// ---- VISUs/v_byte.TcVIS
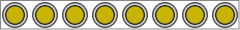
VISUALIZATION v_byte  // 240x30
VAR_IN_OUT
	iNum : INT;
END_VAR
    Lamp1 (0,0 30x30), variable: GVL.stByte.arByte[iNum].Ch[0], style: Lamp-Lamp1-Yellow
    Lamp1 (30,0 30x30), variable: GVL.stByte.arByte[iNum].Ch[1], style: Lamp-Lamp1-Yellow
    Lamp1 (60,0 30x30), variable: GVL.stByte.arByte[iNum].Ch[2], style: Lamp-Lamp1-Yellow
    Lamp1 (90,0 30x30), variable: GVL.stByte.arByte[iNum].Ch[3], style: Lamp-Lamp1-Yellow
    Lamp1 (120,0 30x30), variable: GVL.stByte.arByte[iNum].Ch[4], style: Lamp-Lamp1-Yellow
    Lamp1 (150,0 30x30), variable: GVL.stByte.arByte[iNum].Ch[5], style: Lamp-Lamp1-Yellow
    Lamp1 (180,0 30x30), variable: GVL.stByte.arByte[iNum].Ch[6], style: Lamp-Lamp1-Yellow
    Lamp1 (210,0 30x30), variable: GVL.stByte.arByte[iNum].Ch[7], style: Lamp-Lamp1-Yellow
END_VISUALIZATION

// ---- VISUs/v_IO_ReM.TcVIS
VISUALIZATION v_IO_ReM  // 2048x1080
END_VISUALIZATION

// ---- VISUs/v_rem_0.TcVIS
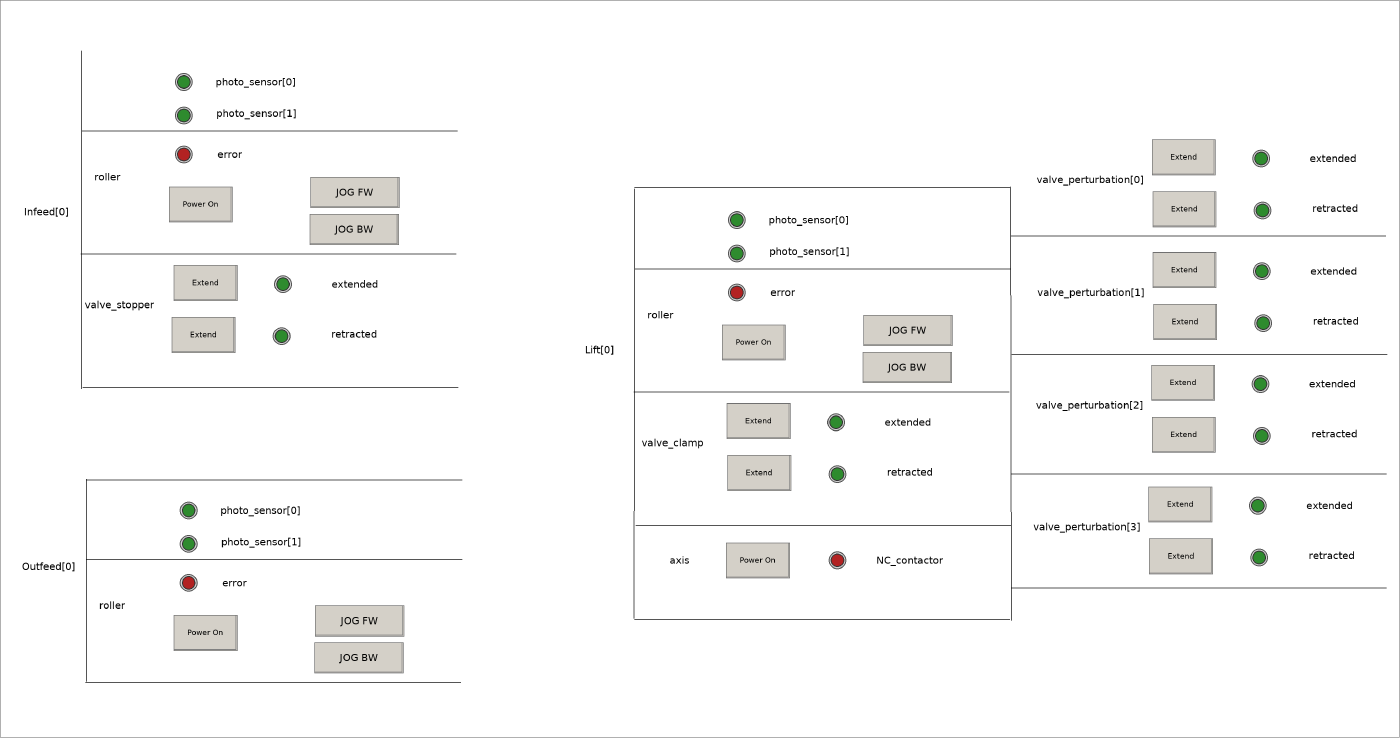
VISUALIZATION v_rem_0  // 2048x1080
VAR_IN_OUT
	dIO_ReM		: Replenishment_Module;
END_VAR
    Lamp1 (254,105 30x30), variable: dIO_ReM.infeed[0].photo_sensor[0].debounced_input.Q, style: Lamp-Lamp1-Green
    Lamp1 (254,154 30x30), variable: dIO_ReM.infeed[0].photo_sensor[1].debounced_input.Q, style: Lamp-Lamp1-Green
    Label (308,107 132x26), "photo_sensor[0]"
    Label (309,153 132x26), "photo_sensor[1]"
    Label (28,297 80x26), "Infeed[0]"
    Lamp1 (254,211 30x30), variable: dIO_ReM.infeed[0].roller.err, style: Lamp-Lamp1-Red
    Label (270,213 132x26), "error"
    Label (91,246 132x26), "roller"
    Line (120,191) (669,191)
    Line (119,74) (119,569)
    Label (109,433 132x26), "valve_stopper"
    Button (454,259 130x45), "JOG FW", colour toggle: dIO_ReM.infeed[0].roller.forward
        OnMouseDown: execute { dIO_ReM.infeed[0].roller.forward := TRUE; }
        OnMouseUp: execute { dIO_ReM.infeed[0].roller.forward := FALSE; }
    Button (453,313 130x45), "JOG BW", colour toggle: dIO_ReM.infeed[0].roller.backward
        OnMouseDown: execute { dIO_ReM.infeed[0].roller.backward := TRUE; }
        OnMouseUp: execute { dIO_ReM.infeed[0].roller.backward := FALSE; }
    Button (247,273 93x52), "Power On", colour toggle: dIO_ReM.infeed[0].roller.Power
        toggle dIO_ReM.infeed[0].roller.Power
    Button (254,388 93x52), "Extend", colour toggle: dIO_ReM.infeed[0].valve_stopper.extend
        OnMouseDown: execute { dIO_ReM.infeed[0].valve_stopper.extend := TRUE; dIO_ReM.infeed[0].valve_stopper.retract := FALSE; }
    Button (251,464 93x52), "Extend", colour toggle: dIO_ReM.infeed[0].valve_stopper.retract
        OnMouseDown: execute { dIO_ReM.infeed[0].valve_stopper.extend := FALSE; dIO_ReM.infeed[0].valve_stopper.retract := TRUE; }
    Lamp1 (399,401 30x30), variable: dIO_ReM.infeed[0].valve_stopper.extended, style: Lamp-Lamp1-Green
    Lamp1 (397,477 30x30), variable: dIO_ReM.infeed[0].valve_stopper.retracted, style: Lamp-Lamp1-Green
    Label (453,403 132x26), "extended"
    Label (452,476 132x26), "retracted"
    Line (118,371) (667,371)
    Line (121,567) (670,567)
    Lamp1 (261,732 30x30), variable: dIO_ReM.outfeed[0].photo_sensor[0].debounced_input.Q, style: Lamp-Lamp1-Green
    Lamp1 (261,781 30x30), variable: dIO_ReM.outfeed[0].photo_sensor[1].debounced_input.Q, style: Lamp-Lamp1-Green
    Label (315,734 132x26), "photo_sensor[0]"
    Label (316,780 132x26), "photo_sensor[1]"
    Label (31,816 80x26), "Outfeed[0]"
    Lamp1 (261,838 30x30), variable: dIO_ReM.outfeed[0].roller.err, style: Lamp-Lamp1-Red
    Label (277,840 132x26), "error"
    Label (98,873 132x26), "roller"
    Line (127,818) (676,818)
    Line (126,701) (126,997)
    Button (461,886 130x45), "JOG FW", colour toggle: dIO_ReM.outfeed[0].roller.forward
        OnMouseDown: execute { dIO_ReM.outfeed[0].roller.forward := TRUE; }
        OnMouseUp: execute { dIO_ReM.outfeed[0].roller.forward := FALSE; }
    Button (460,940 130x45), "JOG BW", colour toggle: dIO_ReM.outfeed[0].roller.backward
        OnMouseDown: execute { dIO_ReM.outfeed[0].roller.backward := TRUE; }
        OnMouseUp: execute { dIO_ReM.outfeed[0].roller.backward := FALSE; }
    Button (254,900 93x52), "Power On", colour toggle: dIO_ReM.outfeed[0].roller.Power
        toggle dIO_ReM.outfeed[0].roller.Power
    Line (125,998) (674,998)
    Line (127,702) (676,702)
    Lamp1 (1063,307 30x30), variable: dIO_ReM.lift[0].photo_sensor[0].debounced_input.Q, style: Lamp-Lamp1-Green
    Lamp1 (1063,356 30x30), variable: dIO_ReM.lift[0].photo_sensor[1].debounced_input.Q, style: Lamp-Lamp1-Green
    Label (1117,309 132x26), "photo_sensor[0]"
    Label (1118,355 132x26), "photo_sensor[1]"
    Label (837,499 80x26), "Lift[0]"
    Lamp1 (1063,413 30x30), variable: dIO_ReM.lift[0].roller.err, style: Lamp-Lamp1-Red
    Label (1079,415 132x26), "error"
    Label (900,448 132x26), "roller"
    Line (929,393) (1478,393)
    Line (928,276) (927,905)
    Label (918,635 132x26), "valve_clamp"
    Button (1263,461 130x45), "JOG FW", colour toggle: dIO_ReM.lift[0].roller.forward
        OnMouseDown: execute { dIO_ReM.lift[0].roller.forward := TRUE; }
        OnMouseUp: execute { dIO_ReM.lift[0].roller.forward := FALSE; }
    Button (1262,515 130x45), "JOG BW", colour toggle: dIO_ReM.lift[0].roller.backward
        OnMouseDown: execute { dIO_ReM.lift[0].roller.backward := TRUE; }
        OnMouseUp: execute { dIO_ReM.lift[0].roller.backward := FALSE; }
    Button (1056,475 93x52), "Power On", colour toggle: dIO_ReM.lift[0].roller.Power
        toggle dIO_ReM.lift[0].roller.Power
    Button (1063,590 93x52), "Extend", colour toggle: dIO_ReM.lift[0].valve_clamp.extend
        OnMouseDown: execute { dIO_ReM.lift[0].valve_clamp.extend := TRUE; dIO_ReM.lift[0].valve_clamp.retract := FALSE; }
    Button (1064,666 93x52), "Extend", colour toggle: dIO_ReM.lift[0].valve_clamp.retract
        OnMouseDown: execute { dIO_ReM.lift[0].valve_clamp.extend := FALSE; dIO_ReM.lift[0].valve_clamp.retract := TRUE; }
    Lamp1 (1208,603 30x30), variable: dIO_ReM.lift[0].valve_clamp.extended, style: Lamp-Lamp1-Green
    Lamp1 (1210,679 30x30), variable: dIO_ReM.lift[0].valve_clamp.retracted, style: Lamp-Lamp1-Green
    Label (1262,605 132x26), "extended"
    Label (1265,678 132x26), "retracted"
    Line (927,573) (1476,573)
    Line (930,769) (1479,769)
    Label (1515,250 160x26), "valve_perturbation[0]"
    Button (1685,204 93x52), "Extend", colour toggle: dIO_ReM.lift[0].valve_perturbation[0].extend
        OnMouseDown: execute { dIO_ReM.lift[0].valve_perturbation[0].extend := TRUE; dIO_ReM.lift[0].valve_perturbation[0].retract := FALSE; }
    Button (1686,280 93x52), "Extend", colour toggle: dIO_ReM.lift[0].valve_perturbation[0].retract
        OnMouseDown: execute { dIO_ReM.lift[0].valve_perturbation[0].extend := FALSE; dIO_ReM.lift[0].valve_perturbation[0].retract := TRUE; }
    Lamp1 (1830,217 30x30), variable: dIO_ReM.lift[0].valve_perturbation[0].extended, style: Lamp-Lamp1-Green
    Lamp1 (1832,293 30x30), variable: dIO_ReM.lift[0].valve_perturbation[0].retracted, style: Lamp-Lamp1-Green
    Label (1884,219 132x26), "extended"
    Label (1887,292 132x26), "retracted"
    Label (1516,415 160x26), "valve_perturbation[1]"
    Button (1686,369 93x52), "Extend", colour toggle: dIO_ReM.lift[0].valve_perturbation[1].extend
        OnMouseDown: execute { dIO_ReM.lift[0].valve_perturbation[1].extend := TRUE; dIO_ReM.lift[0].valve_perturbation[1].retract := FALSE; }
    Button (1687,445 93x52), "Extend", colour toggle: dIO_ReM.lift[0].valve_perturbation[1].retract
        OnMouseDown: execute { dIO_ReM.lift[0].valve_perturbation[1].extend := FALSE; dIO_ReM.lift[0].valve_perturbation[1].retract := TRUE; }
    Lamp1 (1831,382 30x30), variable: dIO_ReM.lift[0].valve_perturbation[1].extended, style: Lamp-Lamp1-Green
    Lamp1 (1833,458 30x30), variable: dIO_ReM.lift[0].valve_perturbation[1].retracted, style: Lamp-Lamp1-Green
    Label (1885,384 132x26), "extended"
    Label (1888,457 132x26), "retracted"
    Label (1514,580 160x26), "valve_perturbation[2]"
    Button (1684,534 93x52), "Extend", colour toggle: dIO_ReM.lift[0].valve_perturbation[2].extend
        OnMouseDown: execute { dIO_ReM.lift[0].valve_perturbation[2].extend := TRUE; dIO_ReM.lift[0].valve_perturbation[2].retract := FALSE; }
    Button (1685,610 93x52), "Extend", colour toggle: dIO_ReM.lift[0].valve_perturbation[2].retract
        OnMouseDown: execute { dIO_ReM.lift[0].valve_perturbation[2].extend := FALSE; dIO_ReM.lift[0].valve_perturbation[2].retract := TRUE; }
    Lamp1 (1829,547 30x30), variable: dIO_ReM.lift[0].valve_perturbation[2].extended, style: Lamp-Lamp1-Green
    Lamp1 (1831,623 30x30), variable: dIO_ReM.lift[0].valve_perturbation[2].retracted, style: Lamp-Lamp1-Green
    Label (1883,549 132x26), "extended"
    Label (1886,622 132x26), "retracted"
    Label (1510,758 160x26), "valve_perturbation[3]"
    Button (1680,712 93x52), "Extend", colour toggle: dIO_ReM.lift[0].valve_perturbation[3].extend
        OnMouseDown: execute { dIO_ReM.lift[0].valve_perturbation[3].extend := TRUE; dIO_ReM.lift[0].valve_perturbation[3].retract := FALSE; }
    Button (1681,788 93x52), "Extend", colour toggle: dIO_ReM.lift[0].valve_perturbation[3].retract
        OnMouseDown: execute { dIO_ReM.lift[0].valve_perturbation[3].extend := FALSE; dIO_ReM.lift[0].valve_perturbation[3].retract := TRUE; }
    Lamp1 (1825,725 30x30), variable: dIO_ReM.lift[0].valve_perturbation[3].extended, style: Lamp-Lamp1-Green
    Lamp1 (1827,801 30x30), variable: dIO_ReM.lift[0].valve_perturbation[3].retracted, style: Lamp-Lamp1-Green
    Label (1879,727 132x26), "extended"
    Label (1882,800 132x26), "retracted"
    Line (1478,273) (1479,908)
    Line (1478,345) (2027,345)
    Line (1480,518) (2029,518)
    Line (1479,693) (2028,693)
    Line (1479,860) (2028,860)
    Line (928,274) (1477,274)
    Line (928,906) (1477,906)
    Label (1265,807 132x26), "NC_contactor"
    Label (928,807 132x26), "axis"
    Button (1062,794 93x52), "Power On", colour toggle: dIO_ReM.lift[0].power_axis
        toggle dIO_ReM.lift[0].power_axis
    Lamp1 (1210,805 30x30), variable: dIO_ReM.lift[0].contactor_axis, style: Lamp-Lamp1-Red
END_VISUALIZATION

// ---- VISUs/v_pm_0.TcVIS
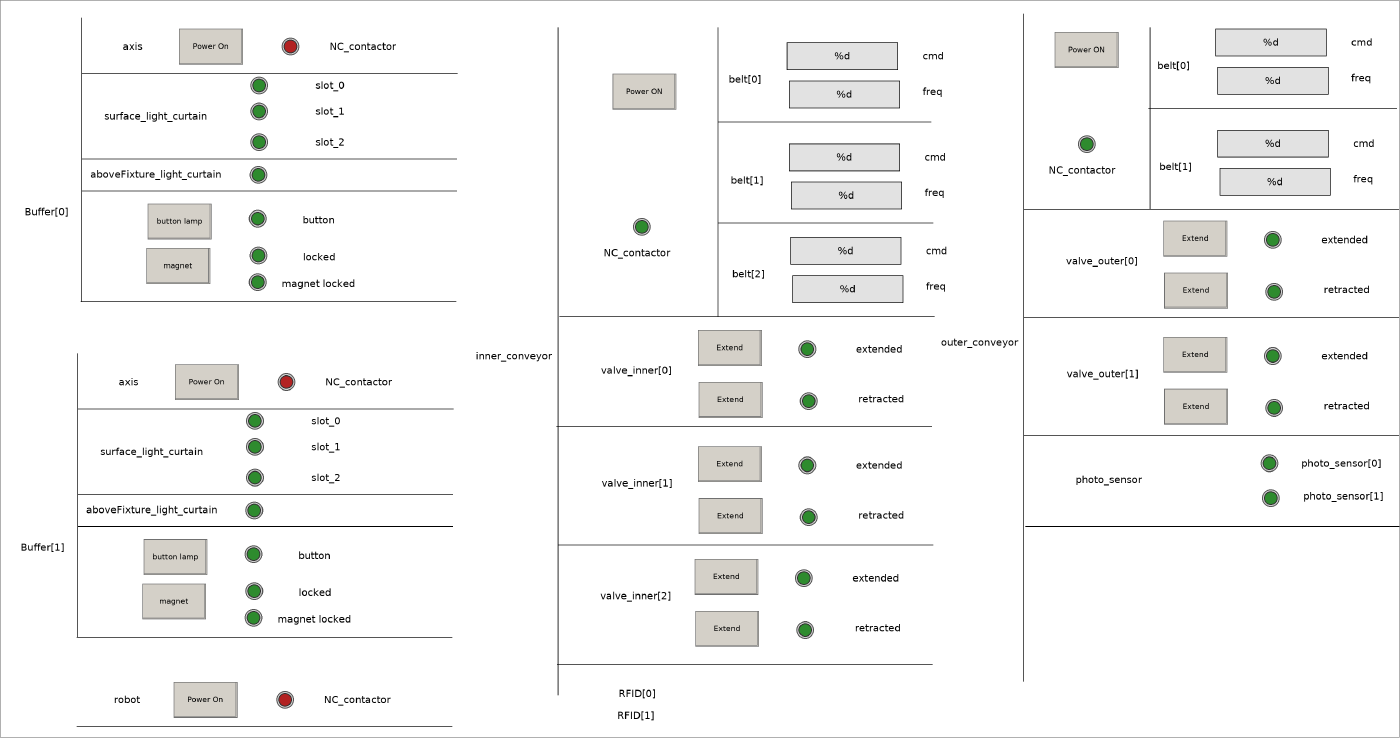
VISUALIZATION v_pm_0  // 2048x1080
VAR_IN_OUT
	dIO_PM		: Picking_Module;
END_VAR
    Lamp1 (364,110 30x30), variable: dIO_PM.buffer[0].surfae_slot_0, style: Lamp-Lamp1-Green
    Label (418,112 130x26), "slot_0"
    Label (28,297 80x26), "Buffer[0]"
    Line (120,107) (669,107)
    Line (119,26) (119,441)
    Line (118,441) (667,441)
    Label (672,508 160x26), "inner_conveyor"
    Line (816,40) (816,1017)
    Label (851,529 160x26), "valve_inner[0]"
    Button (1021,483 93x52), "Extend", colour toggle: dIO_PM.inConv.valve[0].extend
        OnMouseDown: execute { dIO_PM.inConv.valve[0].extend := TRUE; dIO_PM.inConv.valve[0].retract := FALSE; }
    Button (1022,559 93x52), "Extend", colour toggle: dIO_PM.inConv.valve[0].retract
        OnMouseDown: execute { dIO_PM.inConv.valve[0].extend := FALSE; dIO_PM.inConv.valve[0].retract := TRUE; }
    Lamp1 (1166,496 30x30), variable: dIO_PM.inConv.valve[0].extended, style: Lamp-Lamp1-Green
    Lamp1 (1168,572 30x30), variable: dIO_PM.inConv.valve[0].retracted, style: Lamp-Lamp1-Green
    Label (1220,498 132x26), "extended"
    Label (1223,571 132x26), "retracted"
    Label (852,694 160x26), "valve_inner[1]"
    Label (850,859 160x26), "valve_inner[2]"
    Line (814,624) (1363,624)
    Line (816,797) (1365,797)
    Line (815,972) (1364,972)
    Label (465,55 132x26), "NC_contactor"
    Label (128,55 132x26), "axis"
    Button (262,42 93x52), "Power On", colour toggle: dIO_PM.buffer[0].power_axis
        toggle dIO_PM.buffer[0].power_axis
    Lamp1 (410,53 30x30), variable: dIO_PM.buffer[0].contractor_axis, style: Lamp-Lamp1-Red
    Label (128,157 200x26), "surface_light_curtain"
    Label (418,150 130x26), "slot_1"
    Lamp1 (364,148 30x30), variable: dIO_PM.buffer[0].surfae_slot_1, style: Lamp-Lamp1-Green
    Label (418,195 130x26), "slot_2"
    Lamp1 (364,193 30x30), variable: dIO_PM.buffer[0].surfae_slot_2, style: Lamp-Lamp1-Green
    Label (128,242 200x26), "aboveFixture_light_curtain"
    Lamp1 (363,241 30x30), variable: dIO_PM.buffer[0].above_fixture_light_curtain, style: Lamp-Lamp1-Green
    Line (119,232) (668,232)
    Line (119,279) (668,279)
    Label (406,309 120x26), "button"
    Lamp1 (362,305 30x30), variable: dIO_PM.buffer[0].button, style: Lamp-Lamp1-Green
    Button (216,298 93x52), "button lamp", colour toggle: dIO_PM.buffer[0].lamp_button
        toggle dIO_PM.buffer[0].lamp_button
    Button (214,363 93x52), "magnet", colour toggle: dIO_PM.buffer[0].magnet
        toggle dIO_PM.buffer[0].magnet
    Label (407,363 120x26), "locked"
    Lamp1 (363,359 30x30), variable: dIO_PM.buffer[0].locked, style: Lamp-Lamp1-Green
    Label (406,402 120x26), "magnet locked"
    Lamp1 (362,398 30x30), variable: dIO_PM.buffer[0].magnet_locked, style: Lamp-Lamp1-Green
    Lamp1 (358,601 30x30), variable: dIO_PM.buffer[1].surfae_slot_0, style: Lamp-Lamp1-Green
    Label (412,603 130x26), "slot_0"
    Label (22,788 80x26), "Buffer[1]"
    Line (114,598) (663,598)
    Line (113,517) (113,932)
    Line (112,932) (661,932)
    Label (459,546 132x26), "NC_contactor"
    Label (122,546 132x26), "axis"
    Button (256,533 93x52), "Power On", colour toggle: dIO_PM.buffer[1].power_axis
        toggle dIO_PM.buffer[1].power_axis
    Lamp1 (404,544 30x30), variable: dIO_PM.buffer[1].contractor_axis, style: Lamp-Lamp1-Red
    Label (122,648 200x26), "surface_light_curtain"
    Label (412,641 130x26), "slot_1"
    Lamp1 (358,639 30x30), variable: dIO_PM.buffer[1].surfae_slot_1, style: Lamp-Lamp1-Green
    Label (412,686 130x26), "slot_2"
    Lamp1 (358,684 30x30), variable: dIO_PM.buffer[1].surfae_slot_2, style: Lamp-Lamp1-Green
    Label (122,733 200x26), "aboveFixture_light_curtain"
    Lamp1 (357,732 30x30), variable: dIO_PM.buffer[1].above_fixture_light_curtain, style: Lamp-Lamp1-Green
    Line (113,723) (662,723)
    Line (113,770) (662,770)
    Label (400,800 120x26), "button"
    Lamp1 (356,796 30x30), variable: dIO_PM.buffer[1].button, style: Lamp-Lamp1-Green
    Button (210,789 93x52), "button lamp", colour toggle: dIO_PM.buffer[0].lamp_button
        toggle dIO_PM.buffer[1].lamp_button
    Button (208,854 93x52), "magnet", colour toggle: dIO_PM.buffer[1].magnet
        toggle dIO_PM.buffer[1].magnet
    Label (401,854 120x26), "locked"
    Lamp1 (357,850 30x30), variable: dIO_PM.buffer[1].locked, style: Lamp-Lamp1-Green
    Label (400,893 120x26), "magnet locked"
    Lamp1 (356,889 30x30), variable: dIO_PM.buffer[1].magnet_locked, style: Lamp-Lamp1-Green
    Line (112,1063) (661,1063)
    Label (457,1011 132x26), "NC_contactor"
    Label (120,1011 132x26), "robot"
    Button (254,998 93x52), "Power On", colour toggle: dIO_PM.power_robot
        toggle dIO_PM.power_robot
    Lamp1 (402,1009 30x30), variable: dIO_PM.contactor_robot, style: Lamp-Lamp1-Red
    Rectangle (1151,62 162x40), "%d", text variable: dIO_PM.inConv.belt[0].cmd
        OnMouseClick: write the text variable via Default
    Rectangle (1154,118 162x40), "%d", text variable: dIO_PM.inConv.belt[0].freq
        OnMouseClick: write the text variable via Default
    Label (1024,103 132x26), "belt[0]"
    Label (1299,69 132x26), "cmd"
    Label (1298,121 132x26), "freq"
    Line (1050,178) (1362,178)
    Rectangle (1154,210 162x40), "%d", text variable: dIO_PM.inConv.belt[1].cmd
        OnMouseClick: write the text variable via Default
    Rectangle (1157,266 162x40), "%d", text variable: dIO_PM.inConv.belt[1].freq
        OnMouseClick: write the text variable via Default
    Label (1027,251 132x26), "belt[1]"
    Label (1302,217 132x26), "cmd"
    Label (1301,269 132x26), "freq"
    Line (1050,326) (1365,326)
    Rectangle (1156,347 162x40), "%d", text variable: dIO_PM.inConv.belt[2].cmd
        OnMouseClick: write the text variable via Default
    Rectangle (1159,403 162x40), "%d", text variable: dIO_PM.inConv.belt[2].freq
        OnMouseClick: write the text variable via Default
    Label (1029,388 132x26), "belt[2]"
    Label (1304,354 132x26), "cmd"
    Label (1303,406 132x26), "freq"
    Line (818,463) (1367,463)
    Button (1021,653 93x52), "Extend", colour toggle: dIO_PM.inConv.valve[1].extend
        OnMouseDown: execute { dIO_PM.inConv.valve[1].extend := TRUE; dIO_PM.inConv.valve[1].retract := FALSE; }
    Button (1022,729 93x52), "Extend", colour toggle: dIO_PM.inConv.valve[1].retract
        OnMouseDown: execute { dIO_PM.inConv.valve[1].extend := FALSE; dIO_PM.inConv.valve[1].retract := TRUE; }
    Lamp1 (1166,666 30x30), variable: dIO_PM.inConv.valve[1].extended, style: Lamp-Lamp1-Green
    Lamp1 (1168,742 30x30), variable: dIO_PM.inConv.valve[1].retracted, style: Lamp-Lamp1-Green
    Label (1220,668 132x26), "extended"
    Label (1223,741 132x26), "retracted"
    Button (1016,818 93x52), "Extend", colour toggle: dIO_PM.inConv.valve[2].extend
        OnMouseDown: execute { dIO_PM.inConv.valve[2].extend := TRUE; dIO_PM.inConv.valve[2].retract := FALSE; }
    Button (1017,894 93x52), "Extend", colour toggle: dIO_PM.inConv.valve[2].retract
        OnMouseDown: execute { dIO_PM.inConv.valve[2].extend := FALSE; dIO_PM.inConv.valve[2].retract := TRUE; }
    Lamp1 (1161,831 30x30), variable: dIO_PM.inConv.valve[2].extended, style: Lamp-Lamp1-Green
    Lamp1 (1163,907 30x30), variable: dIO_PM.inConv.valve[2].retracted, style: Lamp-Lamp1-Green
    Label (1215,833 132x26), "extended"
    Label (1218,906 132x26), "retracted"
    Label (852,1002 160x26), "RFID[0]"
    Label (850,1034 160x26), "RFID[1]"
    Label (1353,488 160x26), "outer_conveyor"
    Line (1497,20) (1497,997)
    Label (1532,369 160x26), "valve_outer[0]"
    Button (1702,323 93x52), "Extend", colour toggle: dIO_PM.outConv.valve[0].extend
        OnMouseDown: execute { dIO_PM.outConv.valve[0].extend := TRUE; dIO_PM.outConv.valve[0].retract := FALSE; }
    Button (1703,399 93x52), "Extend", colour toggle: dIO_PM.outConv.valve[0].retract
        OnMouseDown: execute { dIO_PM.outConv.valve[0].extend := FALSE; dIO_PM.outConv.valve[0].retract := TRUE; }
    Lamp1 (1847,336 30x30), variable: dIO_PM.outConv.valve[0].extended, style: Lamp-Lamp1-Green
    Lamp1 (1849,412 30x30), variable: dIO_PM.outConv.valve[0].retracted, style: Lamp-Lamp1-Green
    Label (1901,338 132x26), "extended"
    Label (1904,411 132x26), "retracted"
    Label (1533,534 160x26), "valve_outer[1]"
    Line (1498,464) (2047,464)
    Line (1497,637) (2046,637)
    Line (1500,770) (2049,770)
    Rectangle (1778,42 162x40), "%d", text variable: dIO_PM.outConv.belt[0].cmd
        OnMouseClick: write the text variable via Default
    Rectangle (1781,98 162x40), "%d", text variable: dIO_PM.outConv.belt[0].freq
        OnMouseClick: write the text variable via Default
    Label (1651,83 132x26), "belt[0]"
    Label (1926,49 132x26), "cmd"
    Label (1925,101 132x26), "freq"
    Line (1680,158) (2043,158)
    Rectangle (1781,190 162x40), "%d", text variable: dIO_PM.outConv.belt[1].cmd
        OnMouseClick: write the text variable via Default
    Rectangle (1784,246 162x40), "%d", text variable: dIO_PM.outConv.belt[1].freq
        OnMouseClick: write the text variable via Default
    Label (1654,231 132x26), "belt[1]"
    Label (1929,197 132x26), "cmd"
    Label (1928,249 132x26), "freq"
    Line (1497,306) (2046,306)
    Button (1702,493 93x52), "Extend", colour toggle: dIO_PM.outConv.valve[1].extend
        OnMouseDown: execute { dIO_PM.outConv.valve[1].extend := TRUE; dIO_PM.outConv.valve[1].retract := FALSE; }
    Button (1703,569 93x52), "Extend", colour toggle: dIO_PM.outConv.valve[1].retract
        OnMouseDown: execute { dIO_PM.outConv.valve[1].extend := FALSE; dIO_PM.outConv.valve[1].retract := TRUE; }
    Lamp1 (1847,506 30x30), variable: dIO_PM.outConv.valve[1].extended, style: Lamp-Lamp1-Green
    Lamp1 (1849,582 30x30), variable: dIO_PM.outConv.valve[1].retracted, style: Lamp-Lamp1-Green
    Label (1901,508 132x26), "extended"
    Label (1904,581 132x26), "retracted"
    Lamp1 (1842,663 30x30), variable: dIO_PM.outConv.photo_sensor[0], style: Lamp-Lamp1-Green
    Lamp1 (1844,714 30x30), variable: dIO_PM.outConv.photo_sensor[1], style: Lamp-Lamp1-Green
    Label (1896,665 132x26), "photo_sensor[0]"
    Label (1899,713 132x26), "photo_sensor[1]"
    Label (1542,689 160x26), "photo_sensor"
    Line (1050,40) (1050,463)
    Button (896,108 93x52), "Power ON", colour toggle: dIO_PM.power_inConv
        toggle dIO_PM.power_inConv
    Lamp1 (924,317 30x30), variable: dIO_PM.contactor_inConv, style: Lamp-Lamp1-Green
    Label (866,357 132x26), "NC_contactor"
    Line (1682,40) (1682,306)
    Button (1543,47 93x52), "Power ON", colour toggle: dIO_PM.power_outConv
        toggle dIO_PM.power_outConv
    Lamp1 (1575,196 30x30), variable: dIO_PM.contactor_outConv, style: Lamp-Lamp1-Green
    Label (1517,236 132x26), "NC_contactor"
END_VISUALIZATION

// ---- VISUs/v_rem_1.TcVIS
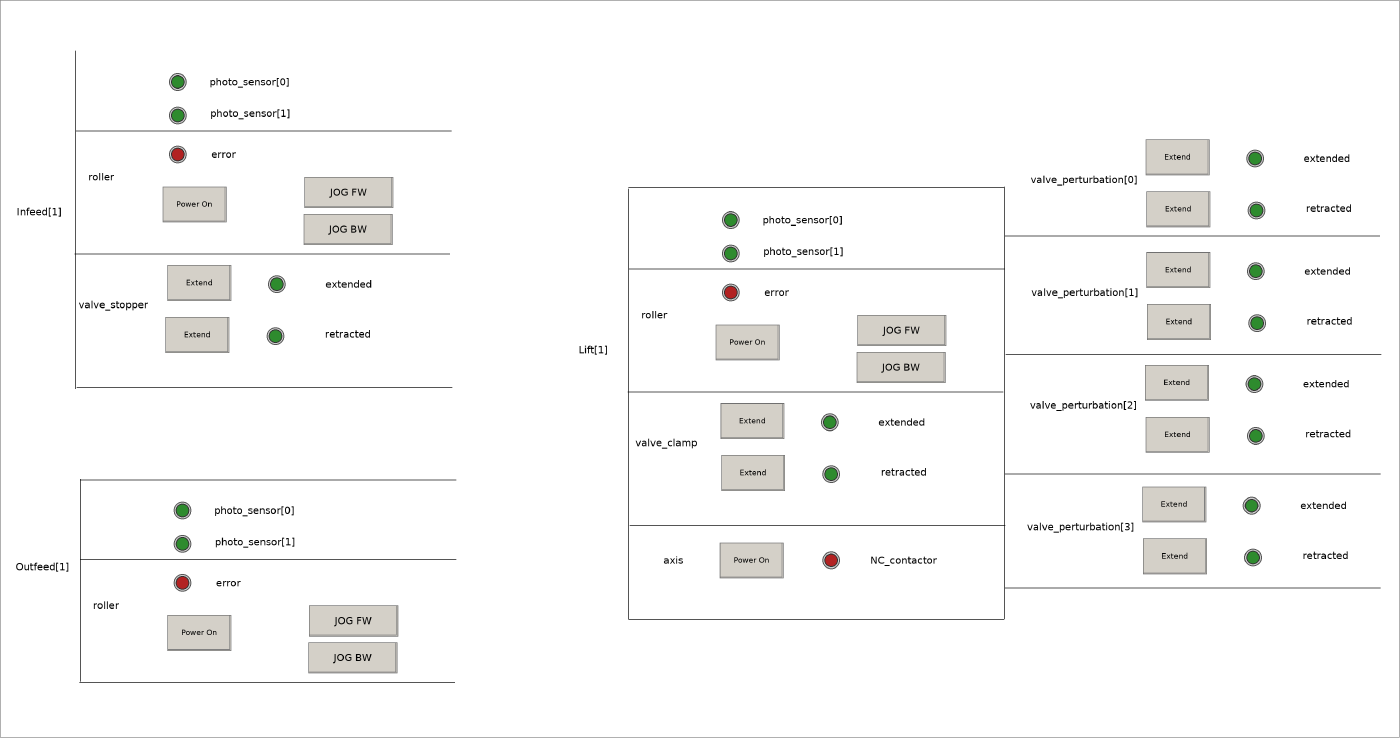
VISUALIZATION v_rem_1  // 2048x1080
VAR_IN_OUT
	dIO_ReM		: Replenishment_Module;
END_VAR
    Lamp1 (245,105 30x30), variable: dIO_ReM.infeed[1].photo_sensor[0].debounced_input.Q, style: Lamp-Lamp1-Green
    Lamp1 (245,154 30x30), variable: dIO_ReM.infeed[1].photo_sensor[1].debounced_input.Q, style: Lamp-Lamp1-Green
    Label (299,107 132x26), "photo_sensor[0]"
    Label (300,153 132x26), "photo_sensor[1]"
    Label (19,297 77x26), "Infeed[1]"
    Lamp1 (245,211 30x30), variable: dIO_ReM.infeed[1].roller.err, style: Lamp-Lamp1-Red
    Label (261,213 132x26), "error"
    Label (82,246 132x26), "roller"
    Line (111,191) (660,191)
    Line (110,74) (110,569)
    Label (100,433 132x26), "valve_stopper"
    Button (445,259 130x45), "JOG FW", colour toggle: dIO_ReM.infeed[1].roller.forward
        OnMouseDown: execute { dIO_ReM.infeed[1].roller.forward := TRUE; }
        OnMouseUp: execute { dIO_ReM.infeed[1].roller.forward := FALSE; }
    Button (444,313 130x45), "JOG BW", colour toggle: dIO_ReM.infeed[1].roller.backward
        OnMouseDown: execute { dIO_ReM.infeed[1].roller.backward := TRUE; }
        OnMouseUp: execute { dIO_ReM.infeed[1].roller.backward := FALSE; }
    Button (238,273 93x52), "Power On", colour toggle: dIO_ReM.infeed[1].roller.Power
        toggle dIO_ReM.infeed[1].roller.Power
    Button (245,388 93x52), "Extend", colour toggle: dIO_ReM.infeed[1].valve_stopper.extend
        OnMouseDown: execute { dIO_ReM.infeed[1].valve_stopper.extend := TRUE; dIO_ReM.infeed[1].valve_stopper.retract := FALSE; }
    Button (242,464 93x52), "Extend", colour toggle: dIO_ReM.infeed[1].valve_stopper.retract
        OnMouseDown: execute { dIO_ReM.infeed[1].valve_stopper.extend := FALSE; dIO_ReM.infeed[1].valve_stopper.retract := TRUE; }
    Lamp1 (390,401 30x30), variable: dIO_ReM.infeed[1].valve_stopper.extended, style: Lamp-Lamp1-Green
    Lamp1 (388,477 30x30), variable: dIO_ReM.infeed[1].valve_stopper.retracted, style: Lamp-Lamp1-Green
    Label (444,403 132x26), "extended"
    Label (443,476 132x26), "retracted"
    Line (109,371) (658,371)
    Line (112,567) (661,567)
    Lamp1 (252,732 30x30), variable: dIO_ReM.outfeed[1].photo_sensor[0].debounced_input.Q, style: Lamp-Lamp1-Green
    Lamp1 (252,781 30x30), variable: dIO_ReM.outfeed[1].photo_sensor[1].debounced_input.Q, style: Lamp-Lamp1-Green
    Label (306,734 132x26), "photo_sensor[0]"
    Label (307,780 132x26), "photo_sensor[1]"
    Label (22,816 80x27), "Outfeed[1]"
    Lamp1 (252,838 30x30), variable: dIO_ReM.outfeed[1].roller.err, style: Lamp-Lamp1-Red
    Label (268,840 132x26), "error"
    Label (89,873 132x26), "roller"
    Line (118,818) (667,818)
    Line (117,701) (117,997)
    Button (452,886 130x45), "JOG FW", colour toggle: dIO_ReM.outfeed[1].roller.forward
        OnMouseDown: execute { dIO_ReM.outfeed[1].roller.forward := TRUE; }
        OnMouseUp: execute { dIO_ReM.outfeed[1].roller.forward := FALSE; }
    Button (451,940 130x45), "JOG BW", colour toggle: dIO_ReM.outfeed[1].roller.backward
        OnMouseDown: execute { dIO_ReM.outfeed[1].roller.backward := TRUE; }
        OnMouseUp: execute { dIO_ReM.outfeed[1].roller.backward := FALSE; }
    Button (245,900 93x52), "Power On", colour toggle: dIO_ReM.outfeed[1].roller.Power
        toggle dIO_ReM.outfeed[1].roller.Power
    Line (116,998) (665,998)
    Line (118,702) (667,702)
    Lamp1 (1054,307 30x30), variable: dIO_ReM.lift[1].photo_sensor[0].debounced_input.Q, style: Lamp-Lamp1-Green
    Lamp1 (1054,356 30x30), variable: dIO_ReM.lift[1].photo_sensor[1].debounced_input.Q, style: Lamp-Lamp1-Green
    Label (1108,309 132x26), "photo_sensor[0]"
    Label (1109,355 132x26), "photo_sensor[1]"
    Label (828,499 80x26), "Lift[1]"
    Lamp1 (1054,413 30x30), variable: dIO_ReM.lift[1].roller.err, style: Lamp-Lamp1-Red
    Label (1070,415 132x26), "error"
    Label (891,448 132x26), "roller"
    Line (920,393) (1469,393)
    Line (919,276) (919,906)
    Label (909,635 132x26), "valve_clamp"
    Button (1254,461 130x45), "JOG FW", colour toggle: dIO_ReM.lift[1].roller.forward
        OnMouseDown: execute { dIO_ReM.lift[1].roller.forward := TRUE; }
        OnMouseUp: execute { dIO_ReM.lift[1].roller.forward := FALSE; }
    Button (1253,515 130x45), "JOG BW", colour toggle: dIO_ReM.lift[1].roller.backward
        OnMouseDown: execute { dIO_ReM.lift[1].roller.backward := TRUE; }
        OnMouseUp: execute { dIO_ReM.lift[1].roller.backward := FALSE; }
    Button (1047,475 93x52), "Power On", colour toggle: dIO_ReM.lift[1].roller.Power
        toggle dIO_ReM.lift[1].roller.Power
    Button (1054,590 93x52), "Extend", colour toggle: dIO_ReM.lift[1].valve_clamp.extend
        OnMouseDown: execute { dIO_ReM.lift[1].valve_clamp.extend := TRUE; dIO_ReM.lift[1].valve_clamp.retract := FALSE; }
    Button (1055,666 93x52), "Extend", colour toggle: dIO_ReM.lift[1].valve_clamp.retract
        OnMouseDown: execute { dIO_ReM.lift[1].valve_clamp.extend := FALSE; dIO_ReM.lift[1].valve_clamp.retract := TRUE; }
    Lamp1 (1199,603 30x30), variable: dIO_ReM.lift[1].valve_clamp.extended, style: Lamp-Lamp1-Green
    Lamp1 (1201,679 30x30), variable: dIO_ReM.lift[1].valve_clamp.retracted, style: Lamp-Lamp1-Green
    Label (1253,605 132x26), "extended"
    Label (1256,678 132x26), "retracted"
    Line (918,573) (1467,573)
    Line (921,769) (1470,769)
    Label (1506,250 160x26), "valve_perturbation[0]"
    Button (1676,204 93x52), "Extend", colour toggle: dIO_ReM.lift[1].valve_perturbation[0].extend
        OnMouseDown: execute { dIO_ReM.lift[1].valve_perturbation[0].extend := TRUE; dIO_ReM.lift[1].valve_perturbation[0].retract := FALSE; }
    Button (1677,280 93x52), "Extend", colour toggle: dIO_ReM.lift[1].valve_perturbation[0].retract
        OnMouseDown: execute { dIO_ReM.lift[1].valve_perturbation[0].extend := FALSE; dIO_ReM.lift[1].valve_perturbation[0].retract := TRUE; }
    Lamp1 (1821,217 30x30), variable: dIO_ReM.lift[1].valve_perturbation[0].extended, style: Lamp-Lamp1-Green
    Lamp1 (1823,293 30x30), variable: dIO_ReM.lift[1].valve_perturbation[0].retracted, style: Lamp-Lamp1-Green
    Label (1875,219 132x26), "extended"
    Label (1878,292 132x26), "retracted"
    Label (1507,415 160x26), "valve_perturbation[1]"
    Button (1677,369 93x52), "Extend", colour toggle: dIO_ReM.lift[1].valve_perturbation[1].extend
        OnMouseDown: execute { dIO_ReM.lift[1].valve_perturbation[1].extend := TRUE; dIO_ReM.lift[1].valve_perturbation[1].retract := FALSE; }
    Button (1678,445 93x52), "Extend", colour toggle: dIO_ReM.lift[1].valve_perturbation[1].retract
        OnMouseDown: execute { dIO_ReM.lift[1].valve_perturbation[1].extend := FALSE; dIO_ReM.lift[1].valve_perturbation[1].retract := TRUE; }
    Lamp1 (1822,382 30x30), variable: dIO_ReM.lift[1].valve_perturbation[1].extended, style: Lamp-Lamp1-Green
    Lamp1 (1824,458 30x30), variable: dIO_ReM.lift[1].valve_perturbation[1].retracted, style: Lamp-Lamp1-Green
    Label (1876,384 132x26), "extended"
    Label (1879,457 132x26), "retracted"
    Label (1505,580 160x26), "valve_perturbation[2]"
    Button (1675,534 93x52), "Extend", colour toggle: dIO_ReM.lift[1].valve_perturbation[2].extend
        OnMouseDown: execute { dIO_ReM.lift[1].valve_perturbation[2].extend := TRUE; dIO_ReM.lift[1].valve_perturbation[2].retract := FALSE; }
    Button (1676,610 93x52), "Extend", colour toggle: dIO_ReM.lift[1].valve_perturbation[2].retract
        OnMouseDown: execute { dIO_ReM.lift[1].valve_perturbation[2].extend := FALSE; dIO_ReM.lift[1].valve_perturbation[2].retract := TRUE; }
    Lamp1 (1820,547 30x30), variable: dIO_ReM.lift[1].valve_perturbation[2].extended, style: Lamp-Lamp1-Green
    Lamp1 (1822,623 30x30), variable: dIO_ReM.lift[1].valve_perturbation[2].retracted, style: Lamp-Lamp1-Green
    Label (1874,549 132x26), "extended"
    Label (1877,622 132x26), "retracted"
    Label (1501,758 160x26), "valve_perturbation[3]"
    Button (1671,712 93x52), "Extend", colour toggle: dIO_ReM.lift[1].valve_perturbation[3].extend
        OnMouseDown: execute { dIO_ReM.lift[1].valve_perturbation[3].extend := TRUE; dIO_ReM.lift[1].valve_perturbation[3].retract := FALSE; }
    Button (1672,788 93x52), "Extend", colour toggle: dIO_ReM.lift[1].valve_perturbation[3].retract
        OnMouseDown: execute { dIO_ReM.lift[1].valve_perturbation[3].extend := FALSE; dIO_ReM.lift[1].valve_perturbation[3].retract := TRUE; }
    Lamp1 (1816,725 30x30), variable: dIO_ReM.lift[1].valve_perturbation[3].extended, style: Lamp-Lamp1-Green
    Lamp1 (1818,801 30x30), variable: dIO_ReM.lift[1].valve_perturbation[3].retracted, style: Lamp-Lamp1-Green
    Label (1870,727 132x26), "extended"
    Label (1873,800 132x26), "retracted"
    Line (1469,273) (1469,906)
    Line (1469,345) (2018,345)
    Line (1471,518) (2020,518)
    Line (1470,693) (2019,693)
    Line (1470,860) (2019,860)
    Line (919,274) (1468,274)
    Line (919,906) (1468,906)
    Label (1256,807 132x26), "NC_contactor"
    Label (919,807 132x26), "axis"
    Button (1053,794 93x52), "Power On", colour toggle: dIO_ReM.lift[1].power_axis
        toggle dIO_ReM.lift[1].power_axis
    Lamp1 (1201,805 30x30), variable: dIO_ReM.lift[1].contactor_axis, style: Lamp-Lamp1-Red
END_VISUALIZATION
